FUNCTION TryConvert_BYTE_TO_INT : BOOL
VAR_INPUT
	in : BYTE;
	out : REFERENCE TO INT;
END_VAR

out := BYTE_TO_INT(in);
TryConvert_BYTE_TO_INT := TRUE;

END_FUNCTION

(* stored: Version 1.1.0.1, ProductVersion 3.1.4024.12
   POU TryConvert_BYTE_TO_INT: Id {92376eb1-e993-4d61-876f-6e45f02e1949}, SpecialFunc None *)
